FUNCTION_BLOCK PUBLIC ShutDown
VAR_INPUT
	GvlIdentifier : STRING;
END_VAR
VAR_OUTPUT
END_VAR
VAR
END_VAR

IF GvlIdentifier = 'R1' THEN
	R1.RecipeStatus		:= FALSE;
	R1.HeatCoolStatus	:= FALSE;
	R1.StirrerStatus	:= FALSE;
	R1.AbortRecipe		:= FALSE;
END_IF;

END_FUNCTION_BLOCK

(* stored: Version 1.1.0.1, ProductVersion 3.1.4024.4
   POU ShutDown: Id {6414f266-d2c5-48ea-8a8c-61388cd5f609}, SpecialFunc None *)
